FUNCTION_BLOCK SectionDelivery (* Basic Function Block Type *)
  (* Standard: 61499-2 *)
  (* Version 0.0, 9/24/2018, dmidro, nxtControl GmbH, Template *)
  PACKAGE Main;
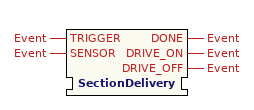
  EVENT_INPUT
    TRIGGER; (* Normal Execution Request *)
    SENSOR;
  END_EVENT
  EVENT_OUTPUT
    DONE; (* Execution Confirmation *)
    DRIVE_ON;
    DRIVE_OFF;
  END_EVENT
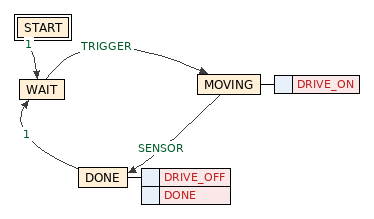
  EC_STATES
    START; (* Initial State *)
    MOVING : -> DRIVE_ON;
    WAIT;
    DONE : -> DRIVE_OFF, -> DONE;
  END_STATES
  EC_TRANSITIONS
    START TO WAIT := 1;
    WAIT TO MOVING := TRIGGER;
    MOVING TO DONE := SENSOR;
    DONE TO WAIT := 1;
  END_TRANSITIONS
  ALGORITHM INIT IN ST: (* Initialization algorithm *)
;
  END_ALGORITHM
  ALGORITHM REQ IN ST: (* Normally executed algorithm *)
;
  END_ALGORITHM
END_FUNCTION_BLOCK
